INTERFACE I_ListComponent Extends I_ListBase

METHOD PUBLIC M_Add : BOOL
VAR_INPUT
	iObject: 	I_Component;
END_VAR
END_METHOD

METHOD PUBLIC M_Request : BOOL
VAR_INPUT
	eRequest:	E_Request;
END_VAR
END_METHOD

METHOD PUBLIC M_Remove : BOOL
VAR_INPUT
	iObject: 	I_Component;
END_VAR
END_METHOD

METHOD PUBLIC M_Find : DINT
VAR_INPUT
	iObject: 	I_Component;
END_VAR
END_METHOD

METHOD PUBLIC M_Index : I_Component
VAR_INPUT
	Index: 	DINT;
END_VAR
END_METHOD

END_INTERFACE

(* stored: Version 1.1.0.1
   Itf I_ListComponent: Id {ab8205a2-82ac-4799-980f-541526123c48}
   Method M_Add: Id {31416f6e-5c2d-4ce2-873c-dc73b1cfa758}
   Method M_Request: Id {4c86b111-cc67-0ae6-0d01-e8bcc72b19a9}
   Method M_Remove: Id {6961a1f7-e686-48a7-b56a-c7aec47523ba}
   Method M_Find: Id {9f020047-7fe7-44c3-b7ac-d3f89fe85683}
   Method M_Index: Id {aa739692-a960-4472-8c48-c3bba57fc92f} *)
